(*~
	<docu>
		<summary>Sample component for inspiration</summary>				
	</docu>
~*)
FUNCTION_BLOCK SampleComponent EXTENDS TcoCore.TcoComponent
VAR
	(*~
		<docu>
			<summary>Counter</summary>
			<remarks>
				> [!IMPORTANT]
				> This member is ignored when rendering.	
			</remarks>			
		</docu>
	~*)
	{attribute clr [RenderIgnore()]}
	_counter : INT;	
END_VAR

VAR
	(*~
		<docu>
			<summary>Counter</summary>
			<remarks>
				> [!IMPORTANT]
				> This member is readonly.
			</remarks>		
		</docu>
	~*)
	{attribute addProperty Name "Add Result"}
	{attribute clr [ReadOnly()]}
	_addResult : INT;
	{attribute addProperty Name "A"}
	_addNumberOne : INT;
	{attribute addProperty Name "B"}
	_addNumberTwo : INT;
END_VAR

VAR	
	_sampleTask : SampleTaskIteration(THIS^);
END_VAR

_addResult := THIS^.AddTwoNumbers(_addNumberOne, _addNumberTwo);
_sampleTask();

(*~
	<docu>
		<summary>Adds two numbers</summary>		
		<returns>Sum of two numbers</returns>
	</docu>
~*)

METHOD AddTwoNumbers : INT
VAR_INPUT
	NumberOne : INT;
	NumberTwo : INT;
END_VAR
AddTwoNumbers := NumberOne + NumberTwo;
END_METHOD

{attribute 'TcRpcEnable'}
METHOD INTERNAL AddTwoNumbersTest : INT
VAR_INPUT
	NumberOne : INT;
	NumberTwo : INT;
END_VAR
AddTwoNumbersTest := THIS^.AddTwoNumbers(NumberOne, NumberTwo);
END_METHOD

METHOD FB_init : BOOL
VAR_INPUT
	bInitRetains : BOOL; // if TRUE, the retain variables are initialized (warm start / cold start)
	bInCopyCode : BOOL;  // if TRUE, the instance afterwards gets moved into the copy code (online change)
	Parent : ITcoObject;
END_VAR
END_METHOD

(*~
	<docu>
		<summary>
			Restores this instance to the Ready state. Can be called explicitly or from within one of the restore mechanisms.	
		</summary>			
	</docu>	
~*)
METHOD  Restore : ITcoRestorable
END_METHOD

(*~
	<docu>
		<summary>
		    Custom service (manual, maintenance) logic.
			This method must be implemented in derived class.
		</summary>			
	</docu>	
~*)
METHOD PROTECTED  ServiceMode
END_METHOD

METHOD WaitForModulo : BOOL
VAR_INPUT
	Modulo : INT;
END_VAR
_counter := _counter + 1;
WaitForModulo := _counter MOD Modulo = 0;
END_METHOD

{attribute 'TcRpcEnable'}
METHOD INTERNAL WaitForModuloTest : BOOL
VAR_INPUT
	Modulo : INT;
END_VAR
WaitForModuloTest := THIS^.WaitForModulo(Modulo);
END_METHOD

END_FUNCTION_BLOCK

(* stored: Version 1.1.0.1, ProductVersion 3.1.4024.9
   POU SampleComponent: Id {faf1774d-d174-0797-11f6-9f36459eabaf}, SpecialFunc None
   Folder _tests: Id {068b66a6-28aa-0256-0f63-8163e3132168}
   Method AddTwoNumbers: Id {93807d61-2d96-0767-2096-405465fd8a7b}
   Method AddTwoNumbersTest: Id {e7ff0940-f609-0d31-2670-486009a10f28}
   Method FB_init: Id {bd2992d8-88c8-0371-17ae-49dd9d4f63cd}
   Method Restore: Id {7579f922-de2b-0342-03e4-f44113979029}
   Method ServiceMode: Id {0687b63b-c7e8-0fff-2d23-03796266c187}
   Method WaitForModulo: Id {04d468d7-88f6-0bbc-2750-023ed3c9d087}
   Method WaitForModuloTest: Id {77bd03ad-6eba-0872-028e-e91ea59ea36d} *)
